VISUALIZATION VISU_State_green_gray  // 12x17
VAR_IN_OUT
	state : BOOL;
END_VAR
    Ellipse (0,5 10x10), colour toggle: state
END_VISUALIZATION

(* stored: Version 1.1.0.1, ProductVersion 3.1.4018.5
   Visu VISU_State_green_gray: Id {35420698-a657-41d8-afb3-74e62faa4958} *)
